Staubli VAL3: getObjectLatch.pgx

public program getObjectLatch(num& x_nLatchedValue[] (dimensions=1), num& x_nError[] (dimensions=1))
  local point l_pPoint
begin
  // This program returns the encoder latched value of the object
  // that have been pushed into the buffer by the detection lib.
  //
  // Input Param
  //  none
  //
  // Output Param
  //  x_nLatchedValue  : encoder latched value of the object
  //  x_nError         : Error code
  //    0 : No error
  //    1 : No data available
  //
  //----------------------------------------------------------------
  //
  x_nError=0
  if nNumbOfUser[nIdxPull]!=0
    x_nLatchedValue=nEncLatchedVal[nIdxPull]
  else
    //* No Object requested
    x_nError=1
    if cfg:bLog==true
      nErrVal[0]=nIdxPull
      call ut:addNumToString(sConvNum+"(getObjectLatch)>>"+sErrMsgList[x_nError],sMsg,"*",nErrVal)
      logMsg(sMsg)
    endIf
  endIf
end
